FUNCTION_BLOCK CSPrint (* Basic Function Block Type *)
  (* Standard: 61499-2 *)
  (* Version 0.2, 2003-12-04, JHC, Rockwell Automation, Renamed for better indexing. *)
  (* Version 0.1, 2002-11-05, JHC, Rockwell Automation, Corrected missing ST element in Algorithm REQ. *)
  (* Version 0.0, 2000-05-30, JHC, Rockwell Automation *)
  (* Compiler header: package fb.rt.cs725; *)
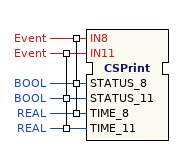
  EVENT_INPUT
    IN8 WITH STATUS_8, TIME_8;
    IN11 WITH STATUS_11, TIME_11;
  END_EVENT
  VAR_INPUT
    STATUS_8 : BOOL;
    STATUS_11 : BOOL;
    TIME_8 : REAL;
    TIME_11 : REAL;
  END_VAR
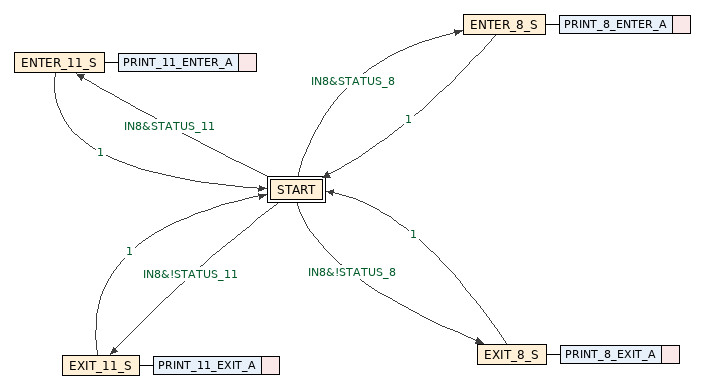
  EC_STATES
    START; (* Initial State *)
    ENTER_8_S : PRINT_8_ENTER_A;
    EXIT_8_S : PRINT_8_EXIT_A;
    ENTER_11_S : PRINT_11_ENTER_A;
    EXIT_11_S : PRINT_11_EXIT_A;
  END_STATES
  EC_TRANSITIONS
    START TO ENTER_8_S := IN8&STATUS_8;
    START TO EXIT_8_S := IN8&!STATUS_8;
    START TO ENTER_11_S := IN8&STATUS_11;
    START TO EXIT_11_S := IN8&!STATUS_11;
    EXIT_11_S TO START := 1;
    EXIT_8_S TO START := 1;
    ENTER_11_S TO START := 1;
    ENTER_8_S TO START := 1;
  END_TRANSITIONS
  ALGORITHM PRINT_11_ENTER_A IN Java:
System.out.println("MULTICAST: Conv 11 entering CS | TIME: "+TIME_11.value);
  END_ALGORITHM
  ALGORITHM PRINT_11_EXIT_A IN Java:
System.out.println("MULTICAST: Conv 11 exiting CS | TIME: "+TIME_11.value);
  END_ALGORITHM
  ALGORITHM PRINT_8_ENTER_A IN Java:
System.out.println("MULTICAST: Conv 8 entering CS | TIME: "+TIME_8.value);
  END_ALGORITHM
  ALGORITHM PRINT_8_EXIT_A IN Java:
System.out.println("MULTICAST: Conv 8 exiting CS | TIME: "+TIME_8.value);
  END_ALGORITHM
END_FUNCTION_BLOCK
